Fanuc KAREL source: CLEAR_SEMA.kl

PROGRAM T
%NOLOCKGROUP
VAR
 v0 : INTEGER
BEGIN
 CLEAR_SEMA(v0)
END T
